{attribute 'qualified_only'}
VAR_GLOBAL
  // ************************General****************************	
  nErrorCodeOKId              : UDINT  := 0;
  nErrorCodeOKStr             : STRING := 'NO ERROR';
  // To high velocity 
  nErrorVelToHigh             : UDINT  := 100;
  sErrorVelToHigh             : STRING := 'MAIN: VELOCITY TO HIGH';
  //Invalid state choosen
  nErrorInvalidState          : UDINT  := 101;
  sErrorInvalidState          : STRING := 'MAIN: Invalid state';
  
  // ************************FB_ModePhase()****************************	
  // No new latched position value have been identified for the last 71 ms (no signal from timing system?)
  nErrorNoLatchId             : UDINT  := 1000;
  sErrorNoLatchStr            : STRING := 'PHASE: NO LATCH FROM DRIVE';
	
  // ************************FB_ModeHome()*****************************
  // The encoder index pulse seems to be lost (a latch have not been identified for the last rev)
  nErrorEncoderLatchLost      : UDINT  := 2000;
  sErrorEncoderLatchLost      : STRING := 'HOME: ENCODER INDEX PULSE LATCH LOST';
  // Deviation found in the latched position values (on index pulse)
  // Could be that encoder pulses are lost or that several index latches occurs per rev.
  nErrorEncoderLatchMissMatch : UDINT  := 2001;
  sErrorEncoderLatchMissMatch : STRING := 'HOME: ENCODER INDEX PULSES POSITION MISSMATCH';
  
  // ************************Indrdradrive*****************************
  nErrorIndraNotReady    : UDINT  := 3000;
  sErrorIndraNotReady    : STRING := 'INDRA: Not ready. Check status of drive (DC-BUS, STO, Tempereature...)';
  nErrorIndraTempToHigh  : UDINT  := 3001;
  sErrorIndraTempToHigh  : STRING := 'INDRA: Motor temperature to high.';
  // Drive not enable
  nErrorNotEnabled       : UDINT  := 3002;
  sErrorNotEnabled       : STRING := 'INDRA: Drive not enabled';
  // Connection lost or re param, need to be re homed
  nErrorNeedHoming       : UDINT  := 3003;
  sErrorNeedHoming       : STRING := 'INDRA: Drive need homing (re param or lost conenction)';
  //Indradrive overheat prewarning
  nErrorIndraOverHeatPrewarning       : UDINT  := 3004;
  sErrorIndraOverHeatPrewarning       : STRING := 'INDRA: Overheat prewarning';
  //Indradrive warning
  nErrorIndraWarning       : UDINT  := 3005;
  sErrorIndraWarning       : STRING := 'INDRA: Warning';
  
END_VAR

(* stored: Version 1.1.0.1, ProductVersion 3.1.4024.6
   GVL GVL_ErrorCodes: Id {2a5675cd-f9a5-4b29-8d57-a071f0a61152} *)
